Staubli VAL3: isActive.pgx

public program isActive(bool& x_bActive, string x_sItem)
begin
  // check it
  if isDefined(saveInOut:cCount[x_sItem])
    x_bActive=saveInOut:cCount[x_sItem].bActive
  elseIf isDefined(saveInOut:aCount[x_sItem])
    x_bActive=(ioStatus(saveInOut:aCount[x_sItem].aAio)>=0)
  else
    // not found
    // toDO
    popUpMsg("value not found: "+x_sItem)
    x_sItem=""
  endIf
end
